{attribute 'linkalways'} 
{attribute 'no_explicit_call' := 'This FB is a CLASS and must be accessed using methods or properties'}
{attribute 'enable_dynamic_creation'}
FUNCTION_BLOCK _TcVnImageInfo EXTENDS StructuredDatatypeBase
VAR
	localData : TcVnImageInfo;
	activeData : REFERENCE TO TcVnImageInfo REF= localData;
	_nImageSize : _ULINT(localData.nImageSize);
	_nWidth : _UDINT(localData.nWidth);
	_nHeight : _UDINT(localData.nHeight);
	_nXPadding : _UINT(localData.nXPadding);
	_nYPadding : _UINT(localData.nYPadding);
	_stPixelFormat : _TcVnPixelFormat();
END_VAR

PROPERTY PUBLIC Address : PVOID
GET
Address := ADR(activeData);
END_GET
END_PROPERTY

METHOD PUBLIC ClearReference
VAR_INPUT
END_VAR
activeData REF= localData;
SetMemberReference();
END_METHOD

METHOD PUBLIC Clone : I_Datatype
VAR
    pClone : POINTER TO _TcVnImageInfo;
END_VAR
pClone := __NEW(_TcVnImageInfo());
pClone^.Value := Value;
Clone := pClone^;
END_METHOD

METHOD FB_init : BOOL
VAR_INPUT
	bInitRetains : BOOL; // if TRUE, the retain variables are initialized (warm start / cold start)
	bInCopyCode : BOOL;  // if TRUE, the instance afterwards gets moved into the copy code (online change)
END_VAR
SetMemberReference();
AddMember('nImageSize',_nImageSize);
AddMember('nWidth',_nWidth);
AddMember('nHeight',_nHeight);
AddMember('nXPadding',_nXPadding);
AddMember('nYPadding',_nYPadding);
AddMember('stPixelFormat',_stPixelFormat);
END_METHOD

PROPERTY PUBLIC Identifier : T_MAXSTRING
GET
Identifier := 'TcVnImageInfo';
END_GET
END_PROPERTY

METHOD PUBLIC MakeReferenceTo
VAR_INPUT
	ReferenceTarget : REFERENCE TO TcVnImageInfo;
END_VAR
activeData REF= ReferenceTarget;
SetMemberReference();
END_METHOD

PROPERTY PUBLIC nHeight : Reference to _UDINT
GET
nHeight REF= _nHeight;
END_GET
END_PROPERTY

PROPERTY PUBLIC nImageSize : Reference to _ULINT
GET
nImageSize REF= _nImageSize;
END_GET
END_PROPERTY

PROPERTY PUBLIC nWidth : Reference to _UDINT
GET
nWidth REF= _nWidth;
END_GET
END_PROPERTY

PROPERTY PUBLIC nXPadding : Reference to _UINT
GET
nXPadding REF= _nXPadding;
END_GET
END_PROPERTY

PROPERTY PUBLIC nYPadding : Reference to _UINT
GET
nYPadding REF= _nYPadding;
END_GET
END_PROPERTY

METHOD PROTECTED SetMemberReference
VAR_INPUT
END_VAR
_nImageSize.MakeReferenceTo(activeData.nImageSize);
_nWidth.MakeReferenceTo(activeData.nWidth);
_nHeight.MakeReferenceTo(activeData.nHeight);
_nXPadding.MakeReferenceTo(activeData.nXPadding);
_nYPadding.MakeReferenceTo(activeData.nYPadding);
_stPixelFormat.MakeReferenceTo(activeData.stPixelFormat);
END_METHOD

PROPERTY PUBLIC Size : UDINT
GET
Size := SIZEOF(activeData);
END_GET
END_PROPERTY

PROPERTY PUBLIC stPixelFormat : Reference to _TcVnPixelFormat
GET
stPixelFormat REF= _stPixelFormat;
END_GET
END_PROPERTY

METHOD TryMakeReferenceTo : BOOL
VAR_INPUT
	Target : I_Datatype;
END_VAR
VAR
	targetAsStruct : I_StructuredDatatype;
	pTargetData : POINTER TO TcVnImageInfo;
END_VAR
IF NOT Target.TryResolveAsStructuredDatatype(targetAsStruct) THEN
	RETURN;
END_IF

IF NOT (targetAsStruct.Identifier = Identifier) THEN
	RETURN;
END_IF

pTargetData := Target.Address;
activeData REF= pTargetData^;
SetMemberReference();
TryMakeReferenceTo := TRUE;
END_METHOD

PROPERTY PUBLIC Value : reference to TcVnImageInfo
GET
Value ref= activeData;
END_GET
END_PROPERTY

END_FUNCTION_BLOCK

(* stored: Version 1.1.0.1, ProductVersion 3.1.4024.12
   POU _TcVnImageInfo: Id {2c5d5a10-3684-0376-3433-17ff4ea4ce21}, SpecialFunc None
   Folder Constructor: Id {6e5007a1-6fe6-0c39-3261-129f6c157fcd}
   Folder Protected: Id {704ed0f1-6e29-0dd0-2f5f-98e0976a76ca}
   Property Address: Id {7206c106-18ff-0fb5-3fe6-85a058bc914a}
   Get Get: Id {a51d28a8-c49a-0b51-26d0-11f18b09bf03}
   Method ClearReference: Id {e58e4960-75aa-08be-11cc-5364e54defaa}
   Method Clone: Id {fc227906-a2ef-0c5f-2dd9-5e5e01f4cde8}
   Method FB_init: Id {171b7e80-3335-0d7b-34d4-def5435953ac}
   Property Identifier: Id {fb33559d-a7f1-00a7-29f7-9b0f36f1fc64}
   Get Get: Id {ebcb9604-6f0a-0c79-16ce-75541ea62fee}
   Method MakeReferenceTo: Id {e811bd81-1db8-0c79-2a33-57052ea160f6}
   Property nHeight: Id {5869b017-f4c5-0b8b-0a78-ba0a3c3dc2c0}
   Get Get: Id {cf4d0ad6-db38-0f06-002d-566894fddef8}
   Property nImageSize: Id {74c20946-9c15-0ef0-273c-34b5e082711c}
   Get Get: Id {e6ce1c0f-d6fa-03d9-1a28-8b90af46d9eb}
   Property nWidth: Id {7a980c4b-79e3-06b3-087f-7f736a3e765e}
   Get Get: Id {307a465c-7cd1-0674-3709-646fda358a89}
   Property nXPadding: Id {52ccc357-ab6d-0601-2d2e-6de05a601438}
   Get Get: Id {676167d0-c37c-026f-211c-0d2e6b956452}
   Property nYPadding: Id {27eb23da-52fe-0285-1c8c-9d4983451012}
   Get Get: Id {874c4d36-0d79-0631-104c-070545430ec7}
   Method SetMemberReference: Id {dc001f08-60a5-0c22-2a01-559af71bca4a}
   Property Size: Id {e8147324-b74b-0006-0e95-dd2b4f034d5c}
   Get Get: Id {9d20fe28-dc77-0695-3dd1-6c0dc6b1852d}
   Property stPixelFormat: Id {10511357-3d9d-069e-0d02-180b2f0971b9}
   Get Get: Id {2434b859-6c6d-01c7-16f2-f6b8d7535dad}
   Method TryMakeReferenceTo: Id {8a5355ad-755a-060d-1093-8030c96fe3a8}
   Property Value: Id {63da58c5-9116-0b86-2897-a385c55398de}
   Get Get: Id {90648104-92f7-0916-27b0-feee5741413a} *)
